INTERFACE I_PLC EXTENDS I_FieldDevice

METHOD M_Comm : BOOL
VAR_INPUT
END_VAR
END_METHOD

END_INTERFACE

(* stored: Version 1.1.0.1, ProductVersion 3.1.4024.15
   Itf I_PLC: Id {3b68cac9-f0b9-4228-8818-339033b4fec3}
   Method M_Comm: Id {9000028c-4bda-4794-9a59-18d66b3b391a} *)
